PROGRAM MAIN
VAR
	PT1T2Parameter :			PT1T2_Parameter_Strukt;
	PID_Parameter :				PID_Parameter_Strukt;
	Modus :						System_Modus_Enum := System_Modus_Enum.System_Init;
	T :							REAL := 0.01;
	PID_1 :						PID_Regler;
	PT1T2_1 :					PT1T2_Prozess;
	r0 :						REAL := 0;	
END_VAR

PT1T2Parameter.K := 10;
PT1T2Parameter.T1 := 0.1;
PT1T2Parameter.T2 := 0.01;

PID_Parameter.Kp := PT1T2Parameter.K;
PID_Parameter.Ti := PT1T2Parameter.T1;
PID_Parameter.Td := PT1T2Parameter.T2;

PID_1(r1 := r0, y1 := PT1T2_1.y, Modus := Modus, Param := PID_Parameter, T := T);
PT1T2_1(u := PID_1.u, Modus := Modus, Param := PT1T2Parameter, T := T);

END_PROGRAM

(* stored: Version 1.1.0.1, ProductVersion 3.1.4024.13
   POU MAIN: Id {688ee701-2e78-402a-871f-5953e56f57cc}, SpecialFunc None *)
